# EPICS substitutions: ek9000App/Db/EL3151.substitutions
file EL3151.template
{       pattern
        {
                TERMINAL,

        }
        {
        }
}
